// TIA Portal V16 export
// export: Created 2025-05-24T14:07:33.1044991Z, ExportSetting WithDefaults, DisplayName Totally Integrated Automation Portal, DisplayVersion V16, DisplayName TIA Portal Version Control Interface, DisplayVersion V16, DisplayName TIA Portal Openness, DisplayVersion V16, DisplayName STEP 7 Professional, DisplayVersion V16, DisplayName STEP 7 Safety, DisplayVersion V16, DisplayName WinCC Advanced, DisplayVersion V16
FUNCTION "3 - Prog. 1" : Void   // FC1, LAD
TITLE = System Program 1
VERSION : 0.1
// DF
// stored: AutoNumber true, IsIECCheckEnabled false, UDAEnableTagReadback false
   VAR_INPUT
      Axis_3_MovePosition1 : Real;
      Axis_3_MovePosition2 : Real;
   END_VAR
   VAR_OUTPUT
      Axis_On_Pos_1 : Bool;
      Axis_On_Pos_2 : Bool;
   END_VAR
   VAR_TEMP
      TempProdCounter : Int;
      Temp_ProductsToProduce : Bool;
      TimerRunning : Bool;
      ProduceContact : Bool;
      Move2Done : Bool;
      SRWals : Bool;
      Move2Busy : Bool;
      SR_Move2 : Bool;
      Move1Busy : Bool;
      P_TRIG_SnrBand : Bool;
      Temp1 : Bool;
      Min_Pos_1 : Real;
      Max_Pos_1 : Real;
      Min_Pos_2 : Real;
      Max_Pos_2 : Real;
      SR_Move3 : Bool;
      SR_Move1 : Bool;
      AxisToRest : Bool;
      SubDone : Bool;
      P_Trig_ProBehWals : Bool;
      ProductsBehindWals : Int;
      ProductBehindWals : Bool;
      AandrukCilindersOut : Bool;
      Retourband_Delayed : Bool;
      BlowOff_Activated : Bool;
      Pos2_Done : Bool;
      Pos1_Done : Bool;
      ToWaitPosition : Bool;
      BlowOffConf : Bool;
      PTrig_Blow : Bool;
      Move2Done_2 : Bool;
      GoToMove2Pos : Bool;
   END_VAR
   VAR_TEMP   // added for the SCL form of the ladder/FBD networks
      _w1 : Bool;
   END_VAR
BEGIN

REGION Network 1: Set Counter on Zero
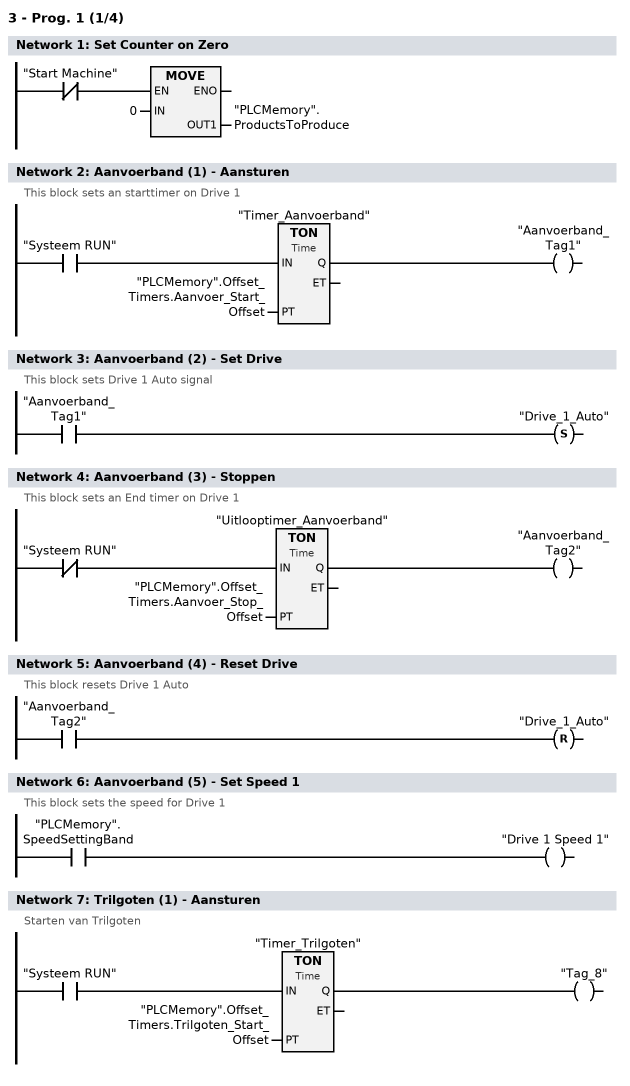
   RUNG wire#powerrail
      I_Contact( "Start Machine" )
      { S7_GenerateENO := "TRUE" } Move(in := 0, out1 => "PLCMemory".ProductsToProduce)
   END_RUNG
   // the same network as SCL:
   IF NOT "Start Machine" THEN "PLCMemory".ProductsToProduce := 0; END_IF;
END_REGION

REGION Network 2: Aanvoerband (1) - Aansturen
   // This block sets an starttimer on Drive 1
   RUNG wire#powerrail
      Contact( "Systeem RUN" )
      { S7_Templates := "time_type := Time" } "Timer_Aanvoerband".TON(pt := "PLCMemory".Offset_Timers.Aanvoer_Start_Offset, et =>)
      Coil( "Aanvoerband_Tag1" )
   END_RUNG
   // the same network as SCL:
   "Timer_Aanvoerband".TON(IN := "Systeem RUN", PT := "PLCMemory".Offset_Timers.Aanvoer_Start_Offset);
   "Aanvoerband_Tag1" := "Timer_Aanvoerband".Q;
END_REGION

REGION Network 3: Aanvoerband (2) - Set Drive
   // This block sets Drive 1 Auto signal
   RUNG wire#powerrail
      Contact( "Aanvoerband_Tag1" )
      S_Coil( "Drive_1_Auto" )
   END_RUNG
   // the same network as SCL:
   IF "Aanvoerband_Tag1" THEN "Drive_1_Auto" := TRUE; END_IF;
END_REGION

REGION Network 4: Aanvoerband (3) - Stoppen
   // This block sets an End timer on Drive 1
   RUNG wire#powerrail
      I_Contact( "Systeem RUN" )
      { S7_Templates := "time_type := Time" } "Uitlooptimer_Aanvoerband".TON(pt := "PLCMemory".Offset_Timers.Aanvoer_Stop_Offset, et =>)
      Coil( "Aanvoerband_Tag2" )
   END_RUNG
   // the same network as SCL:
   "Uitlooptimer_Aanvoerband".TON(IN := NOT "Systeem RUN", PT := "PLCMemory".Offset_Timers.Aanvoer_Stop_Offset);
   "Aanvoerband_Tag2" := "Uitlooptimer_Aanvoerband".Q;
END_REGION

REGION Network 5: Aanvoerband (4) - Reset Drive
   // This block resets Drive 1 Auto
   RUNG wire#powerrail
      Contact( "Aanvoerband_Tag2" )
      R_Coil( "Drive_1_Auto" )
   END_RUNG
   // the same network as SCL:
   IF "Aanvoerband_Tag2" THEN "Drive_1_Auto" := FALSE; END_IF;
END_REGION

REGION Network 6: Aanvoerband (5) - Set Speed 1
   // This block sets the speed for Drive 1
   RUNG wire#powerrail
      Contact( "PLCMemory".SpeedSettingBand )
      Coil( "Drive 1 Speed 1" )
   END_RUNG
   // the same network as SCL:
   "Drive 1 Speed 1" := "PLCMemory".SpeedSettingBand;
END_REGION

REGION Network 7: Trilgoten (1) - Aansturen
   // Starten van Trilgoten
   RUNG wire#powerrail
      Contact( "Systeem RUN" )
      { S7_Templates := "time_type := Time" } "Timer_Trilgoten".TON(pt := "PLCMemory".Offset_Timers.Trilgoten_Start_Offset, et =>)
      Coil( "Tag_8" )
   END_RUNG
   // the same network as SCL:
   "Timer_Trilgoten".TON(IN := "Systeem RUN", PT := "PLCMemory".Offset_Timers.Trilgoten_Start_Offset);
   "Tag_8" := "Timer_Trilgoten".Q;
END_REGION

REGION Network 8: Trilgoten (2) - Set Drive
   // Set drive Trilgoten (Drive 2)
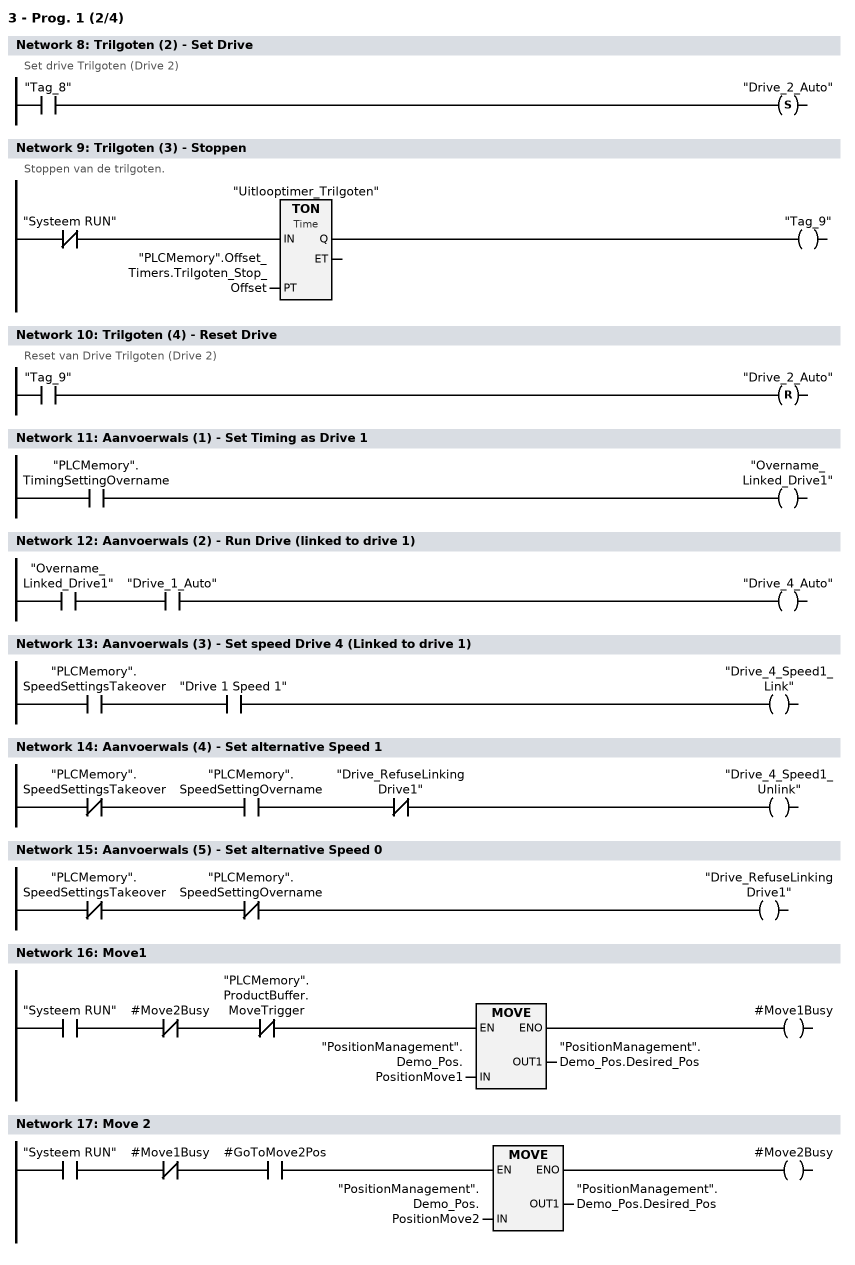
   RUNG wire#powerrail
      Contact( "Tag_8" )
      S_Coil( "Drive_2_Auto" )
   END_RUNG
   // the same network as SCL:
   IF "Tag_8" THEN "Drive_2_Auto" := TRUE; END_IF;
END_REGION

REGION Network 9: Trilgoten (3) - Stoppen
   // Stoppen van de trilgoten.
   RUNG wire#powerrail
      I_Contact( "Systeem RUN" )
      { S7_Templates := "time_type := Time" } "Uitlooptimer_Trilgoten".TON(pt := "PLCMemory".Offset_Timers.Trilgoten_Stop_Offset, et =>)
      Coil( "Tag_9" )
   END_RUNG
   // the same network as SCL:
   "Uitlooptimer_Trilgoten".TON(IN := NOT "Systeem RUN", PT := "PLCMemory".Offset_Timers.Trilgoten_Stop_Offset);
   "Tag_9" := "Uitlooptimer_Trilgoten".Q;
END_REGION

REGION Network 10: Trilgoten (4) - Reset Drive
   // Reset van Drive Trilgoten (Drive 2)
   RUNG wire#powerrail
      Contact( "Tag_9" )
      R_Coil( "Drive_2_Auto" )
   END_RUNG
   // the same network as SCL:
   IF "Tag_9" THEN "Drive_2_Auto" := FALSE; END_IF;
END_REGION

REGION Network 11: Aanvoerwals (1) - Set Timing as Drive 1
   RUNG wire#powerrail
      Contact( "PLCMemory".TimingSettingOvername )
      Coil( "Overname_Linked_Drive1" )
   END_RUNG
   // the same network as SCL:
   "Overname_Linked_Drive1" := "PLCMemory".TimingSettingOvername;
END_REGION

REGION Network 12: Aanvoerwals (2) - Run Drive (linked to drive 1)
   RUNG wire#powerrail
      Contact( "Overname_Linked_Drive1" )
      Contact( "Drive_1_Auto" )
      Coil( "Drive_4_Auto" )
   END_RUNG
   // the same network as SCL:
   "Drive_4_Auto" := "Overname_Linked_Drive1" AND "Drive_1_Auto";
END_REGION

REGION Network 13: Aanvoerwals (3) - Set speed Drive 4 (Linked to drive 1)
   RUNG wire#powerrail
      Contact( "PLCMemory".SpeedSettingsTakeover )
      Contact( "Drive 1 Speed 1" )
      Coil( "Drive_4_Speed1_Link" )
   END_RUNG
   // the same network as SCL:
   "Drive_4_Speed1_Link" := "PLCMemory".SpeedSettingsTakeover AND "Drive 1 Speed 1";
END_REGION

REGION Network 14: Aanvoerwals (4) - Set alternative Speed 1
   RUNG wire#powerrail
      I_Contact( "PLCMemory".SpeedSettingsTakeover )
      Contact( "PLCMemory".SpeedSettingOvername )
      I_Contact( "Drive_RefuseLinkingDrive1" )
      Coil( "Drive_4_Speed1_Unlink" )
   END_RUNG
   // the same network as SCL:
   "Drive_4_Speed1_Unlink" := NOT "PLCMemory".SpeedSettingsTakeover AND "PLCMemory".SpeedSettingOvername AND NOT "Drive_RefuseLinkingDrive1";
END_REGION

REGION Network 15: Aanvoerwals (5) - Set alternative Speed 0
   RUNG wire#powerrail
      I_Contact( "PLCMemory".SpeedSettingsTakeover )
      I_Contact( "PLCMemory".SpeedSettingOvername )
      Coil( "Drive_RefuseLinkingDrive1" )
   END_RUNG
   // the same network as SCL:
   "Drive_RefuseLinkingDrive1" := NOT "PLCMemory".SpeedSettingsTakeover AND NOT "PLCMemory".SpeedSettingOvername;
END_REGION

REGION Network 16: Move1
   RUNG wire#powerrail
      Contact( "Systeem RUN" )
      I_Contact( #Move2Busy )
      I_Contact( "PLCMemory".ProductBuffer.MoveTrigger )
      { S7_GenerateENO := "TRUE" } Move(in := "PositionManagement".Demo_Pos.PositionMove1, out1 => "PositionManagement".Demo_Pos.Desired_Pos)
      Coil( #Move1Busy )
   END_RUNG
   // the same network as SCL:
   // ENO of a box is taken as its EN; it also drops when the box reports an error
   #_w1 := "Systeem RUN" AND NOT #Move2Busy AND NOT "PLCMemory".ProductBuffer.MoveTrigger;
   IF #_w1 THEN
       "PositionManagement".Demo_Pos.Desired_Pos := "PositionManagement".Demo_Pos.PositionMove1;
   END_IF;
   #Move1Busy := #_w1;
END_REGION

REGION Network 17: Move 2
   RUNG wire#powerrail
      Contact( "Systeem RUN" )
      I_Contact( #Move1Busy )
      Contact( #GoToMove2Pos )
      { S7_GenerateENO := "TRUE" } Move(in := "PositionManagement".Demo_Pos.PositionMove2, out1 => "PositionManagement".Demo_Pos.Desired_Pos)
      Coil( #Move2Busy )
   END_RUNG
   // the same network as SCL:
   // ENO of a box is taken as its EN; it also drops when the box reports an error
   #_w1 := "Systeem RUN" AND NOT #Move1Busy AND #GoToMove2Pos;
   IF #_w1 THEN
       "PositionManagement".Demo_Pos.Desired_Pos := "PositionManagement".Demo_Pos.PositionMove2;
   END_IF;
   #Move2Busy := #_w1;
END_REGION

REGION Network 18: Move2 Done
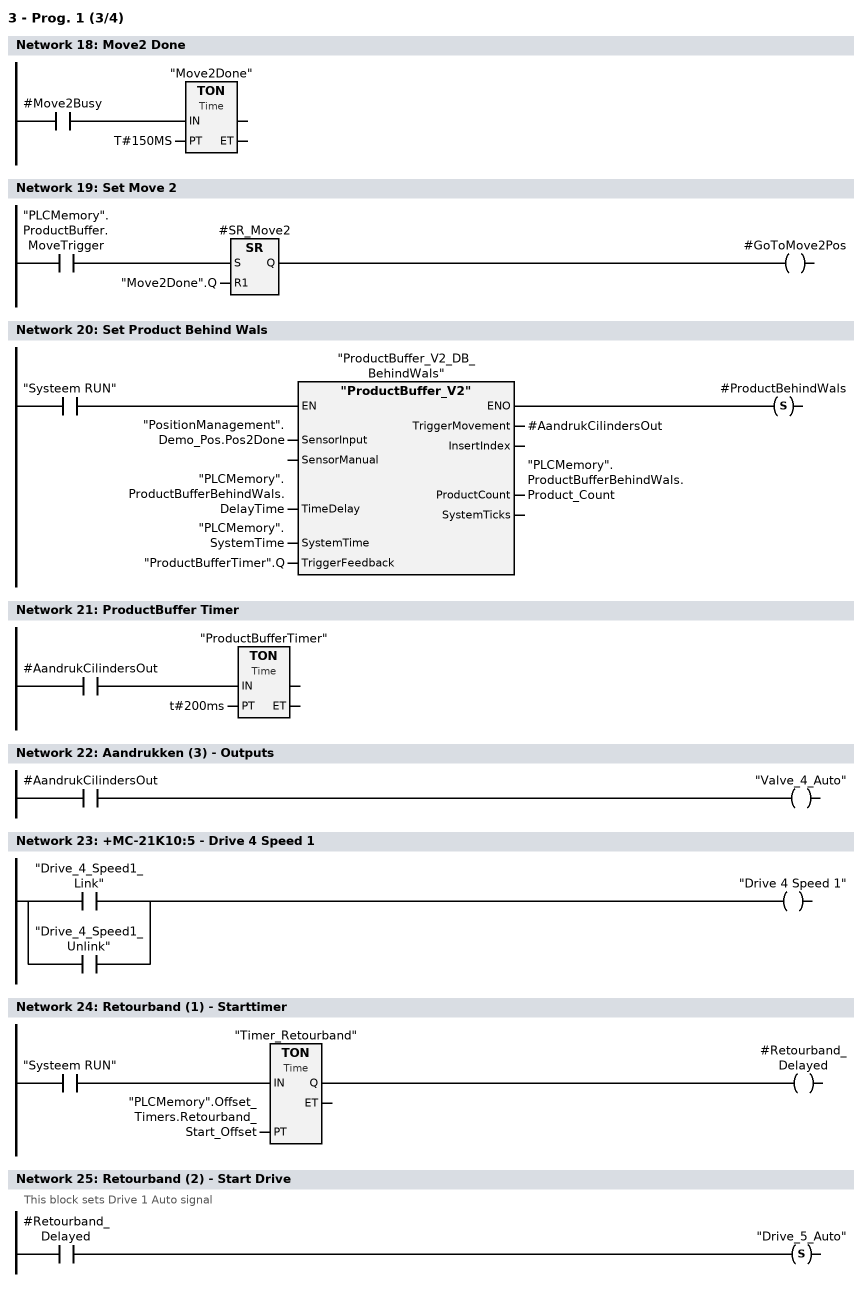
   RUNG wire#powerrail
      Contact( #Move2Busy )
      { S7_Templates := "time_type := Time" } "Move2Done".TON(pt := T#150MS, et =>)
   END_RUNG
   // the same network as SCL:
   "Move2Done".TON(IN := #Move2Busy, PT := T#150MS);
END_REGION

REGION Network 19: Set Move 2
   RUNG wire#powerrail
      Contact( "PLCMemory".ProductBuffer.MoveTrigger )
      S_SR(operand := #SR_Move2, r1 := "Move2Done".Q)
      Coil( #GoToMove2Pos )
   END_RUNG
   // the same network as SCL:
   IF "PLCMemory".ProductBuffer.MoveTrigger THEN
       #SR_Move2 := TRUE;   // SR flip-flop
   END_IF;
   IF "Move2Done".Q THEN #SR_Move2 := FALSE; END_IF;
   #GoToMove2Pos := #SR_Move2;
END_REGION

REGION Network 20: Set Product Behind Wals
   RUNG wire#powerrail
      Contact( "Systeem RUN" )
      "ProductBuffer_V2_DB_BehindWals"(SensorInput := "PositionManagement".Demo_Pos.Pos2Done, SensorManual :=, TimeDelay := "PLCMemory".ProductBufferBehindWals.DelayTime, SystemTime := "PLCMemory".SystemTime, TriggerFeedback := "ProductBufferTimer".Q, TriggerMovement => #AandrukCilindersOut, InsertIndex =>, ProductCount => "PLCMemory".ProductBufferBehindWals.Product_Count, SystemTicks =>)
      S_Coil( #ProductBehindWals )
   END_RUNG
   // the same network as SCL:
   "ProductBuffer_V2_DB_BehindWals"(EN := "Systeem RUN",   // "ProductBuffer_V2"
                           SensorInput := "PositionManagement".Demo_Pos.Pos2Done,
                           TimeDelay := "PLCMemory".ProductBufferBehindWals.DelayTime,
                           SystemTime := "PLCMemory".SystemTime,
                           TriggerFeedback := "ProductBufferTimer".Q,
                           TriggerMovement => #AandrukCilindersOut,
                           ProductCount => "PLCMemory".ProductBufferBehindWals.Product_Count,
                           ENO => #_w1);
   IF #_w1 THEN #ProductBehindWals := TRUE; END_IF;
END_REGION

REGION Network 21: ProductBuffer Timer
   RUNG wire#powerrail
      Contact( #AandrukCilindersOut )
      { S7_Templates := "time_type := Time" } "ProductBufferTimer".TON(pt := t#200ms, et =>)
   END_RUNG
   // the same network as SCL:
   "ProductBufferTimer".TON(IN := #AandrukCilindersOut, PT := t#200ms);
END_REGION

REGION Network 22: Aandrukken (3) - Outputs
   RUNG wire#powerrail
      Contact( #AandrukCilindersOut )
      Coil( "Valve_4_Auto" )
   END_RUNG
   // the same network as SCL:
   "Valve_4_Auto" := #AandrukCilindersOut;
END_REGION

REGION Network 23: +MC-21K10:5 - Drive 4 Speed 1
   RUNG wire#powerrail
      Contact( "Drive_4_Speed1_Link" )
      wire#w1
      Coil( "Drive 4 Speed 1" )
   END_RUNG
   RUNG wire#powerrail
      Contact( "Drive_4_Speed1_Unlink" )
   END_RUNG wire#w1
   // the same network as SCL:
   "Drive 4 Speed 1" := "Drive_4_Speed1_Link" OR "Drive_4_Speed1_Unlink";
END_REGION

REGION Network 24: Retourband (1) - Starttimer
   RUNG wire#powerrail
      Contact( "Systeem RUN" )
      { S7_Templates := "time_type := Time" } "Timer_Retourband".TON(pt := "PLCMemory".Offset_Timers.Retourband_Start_Offset, et =>)
      Coil( #Retourband_Delayed )
   END_RUNG
   // the same network as SCL:
   "Timer_Retourband".TON(IN := "Systeem RUN", PT := "PLCMemory".Offset_Timers.Retourband_Start_Offset);
   #Retourband_Delayed := "Timer_Retourband".Q;
END_REGION

REGION Network 25: Retourband (2) - Start Drive
   // This block sets Drive 1 Auto signal
   RUNG wire#powerrail
      Contact( #Retourband_Delayed )
      S_Coil( "Drive_5_Auto" )
   END_RUNG
   // the same network as SCL:
   IF #Retourband_Delayed THEN "Drive_5_Auto" := TRUE; END_IF;
END_REGION

REGION Network 26: Retourband (3) - Stop Drive
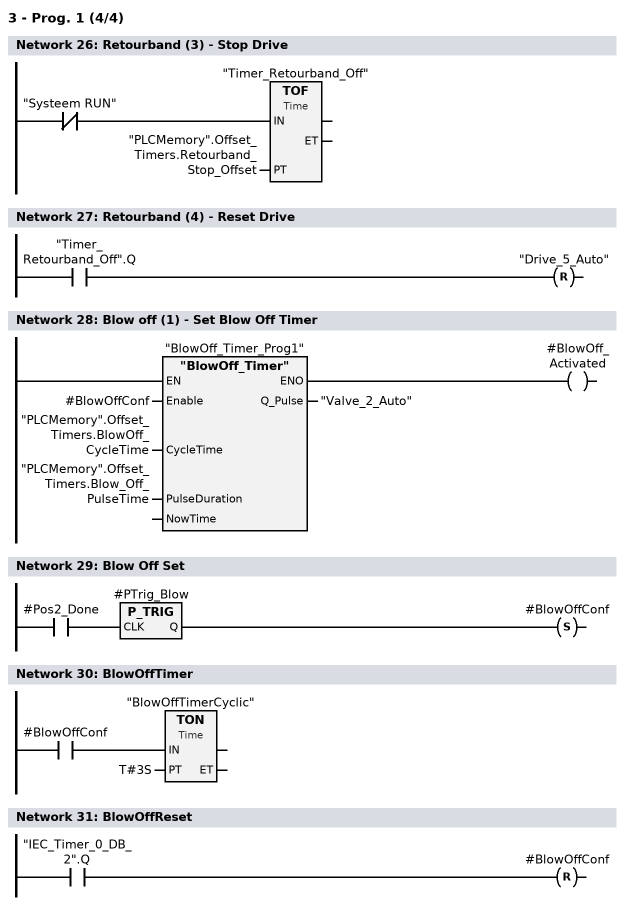
   RUNG wire#powerrail
      I_Contact( "Systeem RUN" )
      { S7_Templates := "time_type := Time" } "Timer_Retourband_Off".TOF(pt := "PLCMemory".Offset_Timers.Retourband_Stop_Offset, et =>)
   END_RUNG
   // the same network as SCL:
   "Timer_Retourband_Off".TOF(IN := NOT "Systeem RUN", PT := "PLCMemory".Offset_Timers.Retourband_Stop_Offset);
END_REGION

REGION Network 27: Retourband (4) - Reset Drive
   RUNG wire#powerrail
      Contact( "Timer_Retourband_Off".Q )
      R_Coil( "Drive_5_Auto" )
   END_RUNG
   // the same network as SCL:
   IF "Timer_Retourband_Off".Q THEN "Drive_5_Auto" := FALSE; END_IF;
END_REGION

REGION Network 28: Blow off (1) - Set Blow Off Timer
   RUNG wire#powerrail
      "BlowOff_Timer_Prog1"(Enable := #BlowOffConf, CycleTime := "PLCMemory".Offset_Timers.BlowOff_CycleTime, PulseDuration := "PLCMemory".Offset_Timers.Blow_Off_PulseTime, NowTime :=, Q_Pulse => "Valve_2_Auto")
      Coil( #BlowOff_Activated )
   END_RUNG
   // the same network as SCL:
   "BlowOff_Timer_Prog1"(Enable := #BlowOffConf,   // "BlowOff_Timer"
                         CycleTime := "PLCMemory".Offset_Timers.BlowOff_CycleTime,
                         PulseDuration := "PLCMemory".Offset_Timers.Blow_Off_PulseTime,
                         Q_Pulse => "Valve_2_Auto",
                         ENO => #_w1);
   #BlowOff_Activated := #_w1;
END_REGION

REGION Network 29: Blow Off Set
   RUNG wire#powerrail
      Contact( #Pos2_Done )
      P_Trig( #PTrig_Blow )
      S_Coil( #BlowOffConf )
   END_RUNG
   // the same network as SCL:
   #_w1 := #Pos2_Done AND NOT #PTrig_Blow;   // rising edge
   #PTrig_Blow := #Pos2_Done;
   IF #_w1 THEN #BlowOffConf := TRUE; END_IF;
END_REGION

REGION Network 30: BlowOffTimer
   RUNG wire#powerrail
      Contact( #BlowOffConf )
      { S7_Templates := "time_type := Time" } "BlowOffTimerCyclic".TON(pt := T#3S, et =>)
   END_RUNG
   // the same network as SCL:
   "BlowOffTimerCyclic".TON(IN := #BlowOffConf, PT := T#3S);
END_REGION

REGION Network 31: BlowOffReset
   RUNG wire#powerrail
      Contact( "IEC_Timer_0_DB_2".Q )
      R_Coil( #BlowOffConf )
   END_RUNG
   // the same network as SCL:
   IF "IEC_Timer_0_DB_2".Q THEN #BlowOffConf := FALSE; END_IF;
END_REGION
END_FUNCTION
